(* CODESYS project preparatorio.project

Project tree, tasks and I/O mapping:
  Device : CODESYS Control Win V3, 3S - Smart Software Solutions GmbH, order no. 305021, version 3.5.11.30
    application Application
      libraries: Standard, * (System)
      task MainTask (cyclic, interval t#20ms, priority 1) calls PLC_PRG
      program PLC_PRG [LD]
      global variables OPCUA
      Symbols
*)

// Device/Application/OPCUA
{attribute 'qualified_only'}
VAR_GLOBAL
	var01: INT;
	var02:INT;
	var03:INT;
	var04:INT;
	
END_VAR

// Device/Application/PLC_PRG
PROGRAM PLC_PRG
VAR
	valor01: INT;
	valor02: INT;
	valor03:INT;
	valor04:INT;
	
	TON_0: TON;
END_VAR
VAR // added by the converter: edge detectors and wires of the graphical bodies
    _w1 : BOOL;
END_VAR

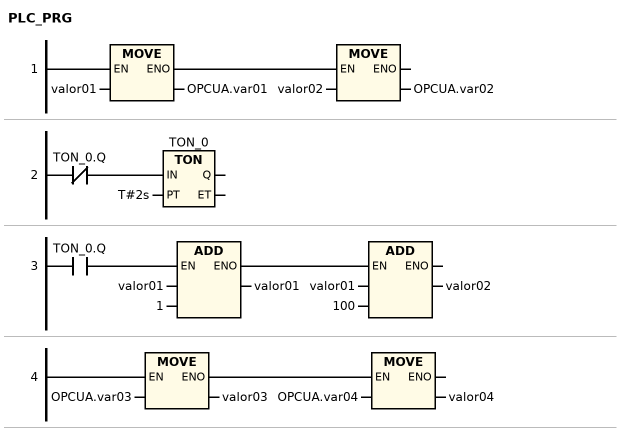
// NETWORK 1
OPCUA.var01 := valor01;
OPCUA.var02 := valor02;

// NETWORK 2
TON_0(IN := NOT TON_0.Q, PT := T#2s); // TON

// NETWORK 3
_w1 := TON_0.Q;
IF _w1 THEN valor01 := valor01 + 1; END_IF
IF _w1 THEN valor02 := valor01 + 100; END_IF

// NETWORK 4
valor03 := OPCUA.var03;
valor04 := OPCUA.var04;

END_PROGRAM
